{attribute clr[Container(Layout.Stack)]}
{attribute clr[Group(Layout.GroupBox)]}
{attribute addProperty PreviousPort "Unknown"}
TYPE EtcSlaveBoxBase_77A0E4A7 EXTENDS EtcSlaveBase_82538BE2 :
STRUCT
END_STRUCT
END_TYPE

(* stored: Version 1.2.0.0, ProductVersion 3.1.4024.11
   DUT EtcSlaveBoxBase_77A0E4A7: Id {cabd467d-6082-444f-b57c-49eb4723e757} *)
